FUNCTION F_GetAmsNetId : T_AmsNetId
VAR_INPUT
   amsNetIdArr : T_AmsNetIdArr;
END_VAR
VAR
   temp : T_AmsNetID;
END_VAR
VAR CONSTANT
   INVALID_LOCAL : T_AmsNetID := '0.0.0.0.0.0';
   LOCAL_NETID : T_AmsNetID := '';
END_VAR

F_GetAmsNetId := F_CreateAmsNetId(amsNetIdArr);

IF F_GetAmsNetId <> INVALID_LOCAL THEN
   RETURN;
END_IF

F_GetAmsNetId := LOCAL_NETID;

END_FUNCTION

(* stored: Version 1.1.0.1, ProductVersion 3.1.4024.9
   POU F_GetAmsNetId: Id {45f5d539-a70c-4ea7-99e7-470e8263da9e}, SpecialFunc None *)
